// TIA Portal V20 export
// export: Created 2025-12-01T14:57:28.9222081Z, ExportSetting None, DisplayName Totally Integrated Automation Portal, DisplayVersion V20 Update 3, DisplayName TIA Portal Openness, DisplayVersion V20 Update 3, DisplayName TIA Portal Version Control Interface, DisplayVersion V20 Update 3, DisplayName STEP 7 Professional, DisplayVersion V20 Update 3, DisplayName STEP 7 Safety, DisplayVersion V20 Update 2, DisplayName WinCC Basic/Comfort/Advanced, DisplayVersion V20 Update 3, DisplayName WinCC Professional, DisplayVersion V20 Update 3, DisplayName WinCC Unified, DisplayVersion V20 Update 3
DATA_BLOCK "DB1604_DB_CBOX04"   // DB1604
AUTHOR : ESTANDAR
NAME : 20160526
VERSION : 3.4
// stored: AutoNumber false, InstanceOfName FB900_CONTROL_ZONA, InstanceOfType FB
"FB900_CONTROL_ZONA"
   // VAR_INPUT
   //    NumZonaUP : UInt;
   //    NumZona : UInt;
   //    MAR_FinReset_DW : Bool;
   //    CONF_Reset_Manual : Bool;
   //    INP_Sel_OffLine : Bool;
   //    INP_Sel_Main : Bool;
   //    INP_Pul_Marcha : Bool;
   //    INP_Pul_Paro : Bool;
   //    INP_Pul_Rearme : Bool;
   //    INP_Pul_TLuces : Bool;
   //    INP_Sel_Automat : Bool;
   //    INP_Sel_Manual : Bool;
   // END_VAR
   // VAR_OUTPUT
   //    L_Verde : Bool;
   //    L_Rojo : Bool;
   //    L_Naranja : Bool;
   //    Sirena : Bool;
   // END_VAR
   // VAR
   //    Toff_Rearme { ExternalAccessible := 'False'; ExternalVisible := 'False'; ExternalWritable := 'False'} : TOF_TIME;
   //    TIM_RetardoMarcha { S7_SetPoint := 'True'} : TON_TIME;
   //    Valor_Cuenta_Reset : UDInt;
   //    Modo_Zona_E0 : Bool;
   //    Modo_Zona_E1 : Bool;
   //    Modo_Zona_E2 : Bool;
   //    Modo_Zona_E3 : Bool;
   //    Modo_Zona_E4 : Bool;
   //    Modo_Zona_E5 : Bool;
   //    S_Paro_Zona : Bool;
   //    S_Marcha_Zona : Bool;
   //    Auto_Zona_E0 : Bool;
   //    Auto_Zona_E1 : Bool;
   //    Auto_Zona_E2 : Bool;
   //    Auto_Zona_E3 : Bool;
   //    Auto_Zona_E4 : Bool;
   //    Auto_Zona_E5 : Bool;
   //    Reset_Zona_E0 : Bool;
   //    Reset_Zona_E1 : Bool;
   //    Reset_Zona_E2 : Bool;
   //    Reset_Zona_E3 : Bool;
   //    Reset_Zona_E4 : Bool;
   //    Reset_Zona_E5 : Bool;
   //    Reset_Zona_E6 : Bool;
   //    Reset_Zona_E7 : Bool;
   //    Mem_PulMarcha_Zona : Bool;
   //    Mem_Error_Zona : Bool;
   //    Mem_Aviso_Error_Zona : Bool;
   //    Mem_Parar_Zona : Bool;
   //    Mem_Reseteo_Zona : Bool;
   //    Mem_PulParo_Zona : Bool;
   //    Mem_Fin_Zona : Bool;
   //    Mem_Fin_Reset_Zona : Bool;
   //    Mem_FP_Rearme : Bool;
   //    Mem_Free2 : Bool;
   //    MemoriaSirena : Bool;
   //    Cuenta_Reset_OK : Bool;
   // END_VAR
BEGIN
END_DATA_BLOCK
